// TwinCAT 3 PLC project Untitled1
// ProgramVersion: 3.1.4024.0
// libraries:
//   Tc2_Standard, * (Beckhoff Automation GmbH)
//   Tc2_System, * (Beckhoff Automation GmbH)
//   Tc3_Module, * (Beckhoff Automation GmbH)
// project tree:
//   DUTs/ E_StudyState.TcDUT
//   GVLs/ GVL_Pomodoro.TcGVL
//   / PlcTask.TcTTO
//   POUs/ CalcBreakTime.TcPOU, MAIN.TcPOU, PRG_StudyTask.TcPOU, PRG_UITask.TcPOU

CONFIGURATION Untitled1
    RESOURCE PLC ON TwinCAT3
        TASK PlcTask(INTERVAL := T#10ms, PRIORITY := 20);
        PROGRAM MAIN WITH PlcTask : MAIN;
    END_RESOURCE
END_CONFIGURATION

// ---- DUTs/E_StudyState.TcDUT
(* DUT: E_StudyState *)

TYPE E_StudyState :
(
    Idle,        (* no timer running *)
    Work,        (* working 25 min *)
    ShortBreak,  (* 5 min break *)
    LongBreak,   (* 15 min break *)
    Paused       (* paused during work *)
);
END_TYPE

// ---- GVLs/GVL_Pomodoro.TcGVL
VAR_GLOBAL
    (* Commands (set from HMI, keyboard, or watch window) *)
    g_bCmdStart      : BOOL := FALSE;   (* rising edge starts / resumes work *)
    g_bCmdPause      : BOOL := FALSE;   (* rising edge pauses work *)
    g_bCmdReset      : BOOL := FALSE;   (* rising edge stops and goes to Idle *)

    (* Process state shared by both tasks *)
    g_eState         : E_StudyState := Idle;
    g_tRemaining     : TIME := T#0s;     (* remaining time in current phase *)
    g_iWorkSessions  : INT := 0;         (* finished work blocks *)
    g_bSessionDone   : BOOL := FALSE;    (* goes TRUE when break finishes *)

    (* “UI outputs” written by Task 2 *)
    g_sStatusText    : STRING(80) := 'Idle';
    g_bLedWork       : BOOL := FALSE;    (* linked to LED or coil *)
    g_bLedBreak      : BOOL := FALSE;    (* linked to LED or coil *)

    (* Just to show result of the function in watch window *)
    g_tLastBreakTime : TIME := T#0s;
END_VAR

// ---- POUs/MAIN.TcPOU
PROGRAM MAIN
VAR
END_VAR

END_PROGRAM

// ---- POUs/CalcBreakTime.TcPOU
FUNCTION CalcBreakTime : TIME
VAR_INPUT
    iWorkSessions : INT;   (* number of finished work blocks *)
END_VAR

(* Long break after every 4th work block, short break otherwise *)
IF (iWorkSessions > 0) AND ((iWorkSessions MOD 4) = 0) THEN
    CalcBreakTime := T#15m;    (* long break *)
ELSE
    CalcBreakTime := T#5m;     (* short break *)
END_IF

END_FUNCTION

// ---- POUs/PRG_StudyTask.TcPOU
PROGRAM PRG_StudyTask
VAR
    tWorkDuration  : TIME := T#25m;
    tBreakDuration : TIME := T#0s;

    fbWorkTimer    : TON;
    fbBreakTimer   : TON;

    bStartEdge     : BOOL;
    bPauseEdge     : BOOL;
    bResetEdge     : BOOL;

    bStartOld      : BOOL;
    bPauseOld      : BOOL;
    bResetOld      : BOOL;
END_VAR

(* Rising edge detection on commands *)
bStartEdge := g_bCmdStart AND NOT bStartOld;
bPauseEdge := g_bCmdPause AND NOT bPauseOld;
bResetEdge := g_bCmdReset AND NOT bResetOld;

bStartOld := g_bCmdStart;
bPauseOld := g_bCmdPause;
bResetOld := g_bCmdReset;

CASE g_eState OF

    (* ================= Idle ================= *)
    Idle:
        (* stop both timers *)
        fbWorkTimer(IN := FALSE, PT := tWorkDuration);
        fbBreakTimer(IN := FALSE, PT := tBreakDuration);

        g_tRemaining   := T#0s;
        g_bSessionDone := FALSE;

        IF bStartEdge THEN
            fbWorkTimer(IN := TRUE, PT := tWorkDuration);
            g_eState := Work;
        END_IF

    (* ================= Work ================= *)
    Work:
        fbWorkTimer(IN := TRUE, PT := tWorkDuration);
        g_tRemaining := tWorkDuration - fbWorkTimer.ET;

        IF bPauseEdge THEN
            fbWorkTimer(IN := FALSE, PT := tWorkDuration);
            g_eState := Paused;

        ELSIF bResetEdge THEN
            fbWorkTimer(IN := FALSE, PT := tWorkDuration);
            g_eState := Idle;

        ELSIF fbWorkTimer.Q THEN
            (* work block finished *)
            fbWorkTimer(IN := FALSE, PT := tWorkDuration);

            g_iWorkSessions := g_iWorkSessions + 1;

            (* === FUNCTION CALL HERE === *)
            tBreakDuration := CalcBreakTime(iWorkSessions := g_iWorkSessions);
            g_tLastBreakTime := tBreakDuration;

            fbBreakTimer(IN := TRUE, PT := tBreakDuration);

            IF tBreakDuration >= T#10m THEN
                g_eState := LongBreak;
            ELSE
                g_eState := ShortBreak;
            END_IF
        END_IF

    (* ========== ShortBreak / LongBreak ========== *)
    ShortBreak,
    LongBreak:
        fbBreakTimer(IN := TRUE, PT := tBreakDuration);
        g_tRemaining := tBreakDuration - fbBreakTimer.ET;

        IF bResetEdge THEN
            fbBreakTimer(IN := FALSE, PT := tBreakDuration);
            g_eState := Idle;

        ELSIF fbBreakTimer.Q THEN
            fbBreakTimer(IN := FALSE, PT := tBreakDuration);
            g_bSessionDone := TRUE;
            g_eState := Idle;
        END_IF

    (* ================= Paused ================= *)
    Paused:
        (* keep timers stopped; remaining time is frozen *)
        fbWorkTimer(IN := FALSE, PT := tWorkDuration);
        fbBreakTimer(IN := FALSE, PT := tBreakDuration);

        IF bStartEdge THEN
            (* resume work *)
            fbWorkTimer(IN := TRUE, PT := tWorkDuration);
            g_eState := Work;
        ELSIF bResetEdge THEN
            g_eState := Idle;
        END_IF

END_CASE

END_PROGRAM

// ---- POUs/PRG_UITask.TcPOU
PROGRAM PRG_UITask
VAR
    fbBlink       : TON;
    tBlinkPeriod  : TIME;
    bLedWorkInt   : BOOL;
END_VAR

(* Choose blink speed based on state *)
CASE g_eState OF
    Idle:
        tBlinkPeriod := T#0s;      (* LED off *)
    Work:
        tBlinkPeriod := T#1s;      (* slow blink while working *)
    ShortBreak:
        tBlinkPeriod := T#500ms;   (* faster blink on short break *)
    LongBreak:
        tBlinkPeriod := T#250ms;   (* very fast blink on long break *)
    Paused:
        tBlinkPeriod := T#2s;      (* slow blink when paused *)
END_CASE

(* Blink logic *)
IF tBlinkPeriod > T#0s THEN
    fbBlink(IN := TRUE, PT := tBlinkPeriod);
    IF fbBlink.Q THEN
        fbBlink(IN := FALSE, PT := tBlinkPeriod);
        bLedWorkInt := NOT bLedWorkInt;
    END_IF
ELSE
    fbBlink(IN := FALSE, PT := tBlinkPeriod);
    bLedWorkInt := FALSE;
END_IF

(* Write UI outputs to global vars *)
g_bLedWork  := bLedWorkInt AND (g_eState = Work);
g_bLedBreak := (g_eState = ShortBreak) OR (g_eState = LongBreak);

CASE g_eState OF
    Idle:       g_sStatusText := 'Idle';
    Work:       g_sStatusText := 'Working';
    ShortBreak: g_sStatusText := 'Short break';
    LongBreak:  g_sStatusText := 'Long break';
    Paused:     g_sStatusText := 'Paused';
END_CASE

END_PROGRAM
